TYPE ST_FSoE_06Byte :
STRUCT
	CMD		: BYTE;
	SafeData1 	: WORD;
	CRC1		: WORD;
	SafeData2 	: WORD;
	CRC2		: WORD;
	SafeData3 	: WORD;
	CRC3		: WORD;
	ConnID		: WORD;
END_STRUCT
END_TYPE

(* stored: Version 1.1.0.1, ProductVersion 3.1.4024.5
   DUT ST_FSoE_06Byte: Id {0429f1c4-959d-45c6-bf5f-26afd99b1105} *)
